PROGRAM MAIN
VAR
	
	hmiAxisSelection: INT := 1; //Not possible to use local hmi variables for array indexes
    afbAxes: ARRAY [1..GVL_APP.nAXIS_NUM] OF FB_Axis;
	
	stAmsNetId	AT %I*	              : AMSNETID;
	nPort	AT %I*                    : WORD;
	nMasterAxisPosition AT %I*        : DINT;
	nMainDriveMarkPosition AT %I*     : DINT;
	nAdditiveTorqueSetpoint    AT %Q* : INT;   // Unit 0.1%  (10=1%)
	dLatchedPosition AT %I*           : DINT;
    fbTemp                            : EL3214_old;
	inputDigSens1 AT %I*              : BOOL;
	inputDigSens2 AT %I*              : BOOL;
	fbModePhase                       : FB_ModePhasing;	 // Phasing Mode
	fbRampVelo                        : FB_RampVelo;
	fbModeVelo                        : FB_ModeVelo;     // Velocity Mode
	fbModePos                         : FB_ModePos;      // Positioning Mode
	fbModeHome                        : FB_ModeHome;     // Homing Mode
	fbIndraDrive                      : fbIndraDrive;    // Control of drive
	
	stCmdEpics                        : ST_CMD_EPICS;    // Control to EPICS 
	stCommands                        : ST_AXIS_COMMAND; // Control to drive
	stStatus                          : ST_AXIS_STATUS;  // Status from drive
	eTargetStateOld                   : TARGET_STATE_MACHINE;
	addStartupTorqueTrigger           : BOOL:=FALSE;
	iTorqueCommandValue  AT %Q*       : INT := 0;
	bApplyTorqueFF                    : BOOL := FALSE;
	nTest: INT;
	
	//hardware
	fbErrorSystem:FB_ErrorSystem;
	fb_s2_EL1809:EL1809;
	fb_s3_EL1809:EL1809;
	fb_s4_EL2819:EL2819;
	fb_s5_EL2819:EL2819;
	fb_s6_EL9505:EL9505;
	fb_s7_EL1252:EL1252;
	fb_s8_EL9410:EL9410;
	fb_s9_EL1252:EL1252;
	fb_s10_EL7201:EL7201;
	fb_s11_EL7201:EL7201;
	fb_s12_EL7201:EL7201;
	fb_s13_EL3214:EL3214;
	fb_s14_EL5021:EL5021;
	fb_s15_EL6695:EL6695;
	fb_s16_EL9410:EL9410;
	fb_s17_EL2032:EL2032;
	fb_s18_EK1110:EK1110;
	fb_s19_IndraDrive:IndraDrive;
	fb_s20_IPOS8020:iPOS8020;
	fb_s21_IPOS8020:iPOS8020;
	fb_s22_IPOS8020:iPOS8020;
	
END_VAR

VAR_INPUT
  stStatEpics                       : ST_STAT_EPICS;   // Status to EPICS
  stHWControlX  : ST_HW_CONTROL_XYZ;
  stHWControlY  : ST_HW_CONTROL_XYZ;
  stHWControlZ  : ST_HW_CONTROL_XYZ;
  stHWControlDev: ST_HW_CONTROL_DEV;
  stHWStatusX   : ST_HW_STATUS_XYZ;
  stHWStatusY   : ST_HW_STATUS_XYZ;
  stHWStatusZ   : ST_HW_STATUS_XYZ;
  stHWStatusDev : ST_HW_STATUS_DEV;
END_VAR

// Check hardware status
ACT_1_Hardware();

// Read Bridge Terminal Inputs
TSCS_Bridge_Inputs();

// Monitor temperature
ACT_2_Temperature();

// Main motor motion
ACT_4_MainDrive();

// Steppers
ACT_5_Steppers();

// Write Bridge Terminal Outputs (incl. test)
TSCS_Bridge_Diagnostic();
TSCS_Bridge_Outputs();

// Error handling
ACT_6_Error();

// Post exe
eTargetStateOld:=stStatEpics.eTargetState;

ACTION ACT_1_Hardware:
// Check state of hardware

// Slave 2 EL1809: General I/O, fuses...
fb_s2_EL1809(ErrorSystem:=fbErrorSystem.pErrorSystem,En:=TRUE,iTerminal_ID:=2);
stHWStatusDev.bEStopOK:=fb_s2_EL1809.bBI_1;                       // s2: ch1: emergency stop ok                 Verify: OK   
stHWStatusDev.bRF02_MainDriveThermalFilterOK:=fb_s2_EL1809.bBI_2; // s2: ch2: rf01 termal braking filter OK..   Verify: Q to Markus: Maybe this should be rd02?
stHWStatusDev.bTA01_TA02_24VSupplyOK:=fb_s2_EL1809.bBI_3;         // s2: ch3: ta01 and ta02 24V power supply OK Verify: OK  
stHWStatusDev.bFC11_Fuse24VOK:=fb_s2_EL1809.bBI_4;                // s2: ch4: fc11 24V fuse OK                   Verify: OK
stHWStatusDev.bFA01_FA02_OvervoltageOK:=fb_s2_EL1809.bBI_5;       // s2: ch5: fa01 and fa02 overvoltage protection OK
stHWStatusDev.bFC01_FuseMainRotationOK:=fb_s2_EL1809.bBI_6;       // s2: ch6: fc01 fuse target wheel motor OK
stHWStatusDev.bFC06_FC07_FuseICSOutletsOK:=fb_s2_EL1809.bBI_7;    // s2: ch7: fc06 and fc07 ICS outlets fuse OK
stHWStatusDev.bFC51_FC52_FC53_FuseUPSOK:=fb_s2_EL1809.bBI_8;      // s2: ch8: fc51, fc52 and fc53 UPS fuses OK (something wrong)

// Slave 3 EL1809: Motion switches (limits)
fb_s3_EL1809(ErrorSystem:=fbErrorSystem.pErrorSystem,En:=TRUE,iTerminal_ID:=3);
main.stHWStatusX.bLimitMax :=fb_s3_EL1809.bBI_1;          // s3: ch1: w02.bg01 stepper x limit max
main.stHWStatusX.bLimitMin :=fb_s3_EL1809.bBI_2;          // s3: ch2: w02.bg02 stepper x limit min
main.stHWStatusX.bLimitMaxMax :=fb_s3_EL1809.bBI_3;       // s3: ch3: w02.bg03 stepper x limit max max
main.stHWStatusX.bLimitMinMin :=fb_s3_EL1809.bBI_4;       // s3: ch4: w02.bg04 stepper x limit min min
main.stHWStatusY.bLimitMax :=fb_s3_EL1809.bBI_5;          // s3: ch5: w02.bg05 stepper y limit max
main.stHWStatusY.bLimitMin :=fb_s3_EL1809.bBI_6;          // s3: ch6: w02.bg06 stepper y limit min
main.stHWStatusY.bLimitMaxMax :=fb_s3_EL1809.bBI_7;       // s3: ch7: w02.bg07 stepper y limit max max
main.stHWStatusY.bLimitMinMin :=fb_s3_EL1809.bBI_8;       // s3: ch8: w02.bg08 stepper y limit min min
main.stHWStatusZ.bLimitMax :=fb_s3_EL1809.bBI_9;          // s3: ch9: w03.bg01 stepper z limit max
main.stHWStatusZ.bLimitMin :=fb_s3_EL1809.bBI_10;         // s3: ch10: w03.bg02 stepper z limit min
main.stHWStatusZ.bLimitMinPark :=fb_s3_EL1809.bBI_11;     // s3: ch11: w03.bg03 stepper z limit min service (lowest switch)
main.stHWStatusZ.bLimitMaxMax :=fb_s3_EL1809.bBI_12;      // s3: ch12: w03.bg04 stepper z limit max max
main.stHWStatusZ.bLimitMinMin :=fb_s3_EL1809.bBI_13;      // s3: ch13: w03.bg05 stepper z limit min min
main.stHWStatusZ.bLimitMinMinPark :=fb_s3_EL1809.bBI_14;  // s3: ch14: w03.bg06 stepper z limit min min service (lowest switch)
main.stHWStatusX.bLimitMinPark:=FALSE;                    // Not used
main.stHWStatusX.bLimitMinMinPark:=FALSE;                 // Not used
main.stHWStatusX.bParkingRangeEnabled:=FALSE;             // Not used;
main.stHWStatusY.bLimitMinPark:=FALSE;                    // Not used
main.stHWStatusY.bLimitMinMinPark:=FALSE;                 // Not used
main.stHWStatusY.bParkingRangeEnabled:=FALSE;             // Not used;

// Slave 4 EL2809: Feed sensors
fb_s4_EL2819(ErrorSystem:=fbErrorSystem.pErrorSystem,En:=TRUE,iTerminal_ID:=4);
stHWControlDev.bRotOmronSensor1Feed:=TRUE;     // s4: ch1: Feed omron sensor 1
stHWControlDev.bRotOmronSensor2Feed:=TRUE;     // s4: ch2: Feed omron sensor 2

// Slave 5 EL2809: Feed switches and brakes
fb_s5_EL2819(ErrorSystem:=fbErrorSystem.pErrorSystem,En:=TRUE,iTerminal_ID:=5);
stHWControlX.bMinMaxFeed:=TRUE;           // s5: ch1: kf05: w02.bg01 w02.bg02 stepper x limit switch max, limit min
//stHWControl.bXBrakeReleaseCmd           // s5: ch2: kf05: w02.ql1: stepper x brake
stHWControlX.bMinMinMaxMaxFeed:=TRUE;     // s5: ch3: kf05: w02.bg03 w02.bg04 stepper x limit switch max max, limit min min
stHWControlY.bMinMaxFeed:=TRUE;           // s5: ch5: kf05: w02.bg05 w02.bg06 stepper y limit switch max, limit min
//stHWControl.bYBrakeReleaseCmd           // s5: ch6: kf05: w02.ql2: stepper y brake
stHWControlY.bMinMinMaxMaxFeed:=TRUE;     // s5: ch7: kf05: w02.bg07 w02.bg08 stepper y limit switch max max, limit min min
stHWControlZ.bMinMaxFeed:=TRUE;           // s5: ch9: kf05: w03.bg01 w03.bg02 w03.bg03  stepper z limit switch max, limit min limit min min (service)
stHWControlZ.bMinMinMaxMaxFeed:=TRUE;     // s5: ch10: kf05: w03.bg04 w03.bg05 w03.bg06  stepper z limit switch max max, limit min min
// Note brakes needs control!!!

// s6: 5V power supply
fb_s6_EL9505(ErrorSystem:=fbErrorSystem.pErrorSystem,En:=TRUE,iTerminal_ID:=6);

// s7: time stamped 5V input from timing system (timing reference pulse 14Hz)
// s7: ch1: kf06. Timing system ref pulse (14Hz). Synch pulse ICS.
fb_s7_EL1252(ErrorSystem:=fbErrorSystem.pErrorSystem,En:=TRUE,iTerminal_ID:=7);

// s8: 24V power supply
fb_s8_EL9410(ErrorSystem:=fbErrorSystem.pErrorSystem,En:=TRUE,iTerminal_ID:=8);

// s9: Omron time stamp 24V
// s9: ch1: w01.bg01 fibre sensor input (home or sector?)
// s9: ch2: w01.bg02 fibre sensor input (home or sector?)
fb_s9_EL1252(ErrorSystem:=fbErrorSystem.pErrorSystem,En:=TRUE,iTerminal_ID:=9);

// s10 ch1: kf09 w02.bg21 Resolver X  
fb_s10_EL7201(ErrorSystem:=fbErrorSystem.pErrorSystem,En:=TRUE,iTerminal_ID:=10);

// s11 ch1: kf10 w02.bg22 Resolver Y
fb_s11_EL7201(ErrorSystem:=fbErrorSystem.pErrorSystem,En:=TRUE,iTerminal_ID:=11);

// s11 ch1: kf11 w03.bg21 Resolver Z
fb_s12_EL7201(ErrorSystem:=fbErrorSystem.pErrorSystem,En:=TRUE,iTerminal_ID:=12);

// s13 EL3214: Temperature inputs X,Y,Z and rotation
fb_s13_EL3214(ErrorSystem:=fbErrorSystem.pErrorSystem,En:=TRUE,iTerminal_ID:=13);
stHWStatusX.fStepperTemp:=INT_TO_LREAL(fb_s13_EL3214.iAI_1)/10; // s13: ch1: kf12 w02.bt01 temperature stepper X PT100
stHWStatusY.fStepperTemp:=INT_TO_LREAL(fb_s13_EL3214.iAI_2)/10; // s13: ch2: kf12 w02.bt02 temperature stepper Y PT100
stHWStatusZ.fStepperTemp:=INT_TO_LREAL(fb_s13_EL3214.iAI_3)/10; // s13: ch3: kf12 w03.bt01 temperature stepper Z PT100
stHWStatusDev.fKF12_RotTemp:=INT_TO_LREAL(fb_s13_EL3214.iAI_4)/10;   // s13: ch4: kf12 Target Main motor Temperature (KTY) (in deg*10)

// s14: Extra encoder (main rotation)
fb_s14_EL5021(ErrorSystem:=fbErrorSystem.pErrorSystem,En:=TRUE,iTerminal_ID:=14);

// s15: Communication to monitoring system
fb_s15_EL6695(ErrorSystem:=fbErrorSystem.pErrorSystem,En:=TRUE,iTerminal_ID:=15);

// s15: 24V power supply
fb_s16_EL9410(ErrorSystem:=fbErrorSystem.pErrorSystem,En:=TRUE,iTerminal_ID:=16);

// s17: MPS com.
fb_s17_EL2032(ErrorSystem:=fbErrorSystem.pErrorSystem,En:=TRUE,iTerminal_ID:=17);

// s1?: Two EL2612 Relay for MPS not in system yet
// s1?: ch1: kf17 Ready for beam
// s1?: ch2: kf17 Beam permit
// s1?: ch3: kf18 Ready for beam
// s1?: ch4: kf18 Beam permit

// s18: extension to drives
fb_s18_EK1110(ErrorSystem:=fbErrorSystem.pErrorSystem,En:=TRUE,iTerminal_ID:=18);

// s19: Main target drive
fb_s19_IndraDrive(ErrorSystem:=fbErrorSystem.pErrorSystem,En:=TRUE,iTerminal_ID:=19);

// s20: Stepper 1
fb_s20_IPOS8020(ErrorSystem:=fbErrorSystem.pErrorSystem,En:=TRUE,iTerminal_ID:=20);

// s21: Stepper 2
fb_s21_IPOS8020(ErrorSystem:=fbErrorSystem.pErrorSystem,En:=TRUE,iTerminal_ID:=21);

// s22: Stepper 3
fb_s22_IPOS8020(ErrorSystem:=fbErrorSystem.pErrorSystem,En:=TRUE,iTerminal_ID:=22);

fbErrorSystem(En:=TRUE);
END_ACTION

ACTION ACT_2_Temperature:
// Function: Monitor tempertures
// Interlock motion on temperatures
// Author: Anders Sandström 2019

stStatEpics.fActTemp:=fb_s13_EL3214.iAI_4/10.0;

// Motor Temperature Monitoring Interlock
IF (stStatEpics.fActTemp >= GVL_Parameters.nMaxMotorTemperature)  OR fbTemp.iAi_Ch1_Stat > 0 THEN
	stCmdEpics.bEnable:= FALSE;
	stCmdEpics.bExecute:= FALSE;
	stStatEpics.nErrorId:=GVL_ErrorCodes.nErrorIndraTempToHigh;
	stStatEpics.sErrorStr:=GVL_ErrorCodes.sErrorIndraTempToHigh;
END_IF
END_ACTION

ACTION ACT_4_MainDrive:

// Enable Axis independent of state (Ensure that drive is ready to enable)
IF stCmdEpics.bEnable THEN
   IF stStatus.bDCBusPresent AND NOT stStatus.bSTOActiveCh1 AND NOT stStatus.bSTOActiveCh2 AND NOT stStatus.bError THEN 
	   stCommands.bEnableAxis :=stCmdEpics.bEnable;
   ELSE
	   stCommands.bEnableAxis := FALSE;
	   stCmdEpics.bExecute := FALSE;
	   stStatEpics.bError:=TRUE;
	   stStatEpics.nErrorId:=GVL_ErrorCodes.nErrorIndraNotReady;
	   stStatEpics.sErrorStr:=GVL_ErrorCodes.sErrorIndraNotReady; 
   END_IF
ELSE
	//Reset enable
    stCommands.bEnableAxis:=stCmdEpics.bEnable;
END_IF

IF stCmdEpics.bExecute THEN
  IF stStatus.bAxisEnabled THEN
    stCommands.bHaltAxis:=stCmdEpics.bExecute;
  ELSE
	stCmdEpics.bExecute:=FALSE;
	stCommands.bHaltAxis:=FALSE;
	stStatEpics.nErrorId:=GVL_ErrorCodes.nErrorNotEnabled;
	stStatEpics.sErrorStr:=GVL_ErrorCodes.sErrorNotEnabled; 
  END_IF
ELSE
  stCommands.bHaltAxis:=stCmdEpics.bExecute;
END_IF

IF NOT stCommands.bEnableAxis THEN
  stCmdEpics.bExecute:=FALSE;
END_IF

stStatEpics.bEnabled:=stStatus.bAxisEnabled;
stCommands.bCmd_ErrorReset:=stCmdEpics.bReset;

stCommands.bCmd_DriveControlledHoming:=FALSE;

// State change
IF stCmdEpics.eTargetStateCmd <> stStatEpics.eTargetState AND NOT stCmdEpics.bexecute AND stStatus.bAxisStandStillStatus THEN
    // Only allow state change if execute is low and at standstill
    stStatEpics.eTargetState:=stCmdEpics.eTargetStateCmd;
END_IF

IF stCmdEpics.fPhaseOffsetMM > GVL_Parameters.fMaxPhaseOffsetMM THEN
	stCmdEpics.fPhaseOffsetMM :=  GVL_Parameters.fMaxPhaseOffsetMM;
END_IF
IF stCmdEpics.fPhaseOffsetMM < GVL_Parameters.fMinPhaseOffsetMM THEN
	stCmdEpics.fPhaseOffsetMM :=  GVL_Parameters.fMinPhaseOffsetMM;
END_IF

stStatEpics.fPhaseOffsetActDeg := stCmdEpics.fPhaseOffsetMM /(GVL_Parameters.fWheelDiameter*pi/360.0);

//nAdditiveTorqueSetpoint:=0;
//IF NOT  stCmdEpics.bExecute THEN
//	addStartupTorqueTrigger:=TRUE;
//END_IF


CASE stStatEpics.eTargetState OF 
	TARGET_STATE_MACHINE.CONSTANT_VELOCITY:
        stCommands.fCommandAcceleration:=GVL_Parameters.fAccDefaultVel;
        stCommands.fCommandDeceleration:=GVL_Parameters.fAccDefaultVel;
		fbModeVelo(
            bExecute:=         stCmdEpics.bExecute,
            bReset:=           stCmdEpics.bReset,
			fVelSet:=          stCmdEpics.fVelSet,
			stStatus:=	       stStatus,	
			stCommands:=       stCommands);
			
			//ramp velocity with selected acceleration
			fbRampVelo(bExecute:=stCmdEpics.bExecute,
              fVelSetIn:=fbModeVelo.fSpeedSetpoint,
              iBlockSampleTimeMicroS:=GVL_Parameters.nTaskSampleTime*1000,
              fVelSetOut:=stCommands.fVelocityCommandValue,
              fVelActIn:=stStatus.fActualVelocity/10);
			  
// add extra torque att startup TEST
		//	IF stStatus.bAxisEnabled AND stCmdEpics.bExecute AND stCmdEpics.fVelSet > 0 THEN
		//		IF stStatus.fActualVelocity/10< stCmdEpics.fVelSet/2 THEN
		//	        nAdditiveTorqueSetpoint:=100;  //Add 10% when under x rpm
		//		ELSIF stStatus.fActualVelocity/10 > stCmdEpics.fVelSet/2 THEN
		//			nAdditiveTorqueSetpoint:=40;
		//		END_IF
		//	END_IF

			
	TARGET_STATE_MACHINE.POSITIONING:
	    stCommands.fCommandAcceleration:=GVL_Parameters.fAccDefaultPos;
        stCommands.fCommandDeceleration:=GVL_Parameters.fAccDefaultPos;

		fbModePos(
            bExecute:=         stCmdEpics.bExecute,
            bReset:=           stCmdEpics.bReset,
			fVelSet:=          stCmdEpics.fVelSet,
			fPosSet:=          stCmdEpics.fPosSet,
			fRefOffset:=       fbModeHome.fActPositionOffset,
			stStatus:=         stStatus,	
			stCommands:=       stCommands);
		
	TARGET_STATE_MACHINE.PHASING:
	    stCommands.fCommandAcceleration:=GVL_Parameters.fAccDefaultVel;
        stCommands.fCommandDeceleration:=GVL_Parameters.fAccDefaultVel;
   		fbModePhase(
			bExecute:=         stCmdEpics.bExecute,
            bReset:=           stCmdEpics.bReset,
			stStatus:=	       stStatus,
			dLatchedPosition:= dLatchedPosition,
			ePhaseType:=       stCmdEpics.ePhaseCntrlAlg,
			ePwmType:=         stCmdEpics.ePhasePwmType,
			stCommands:=       stCommands,
            fPhaseOffsetMM:=   stCmdEpics.fPhaseOffsetMM,
            fRefOffset:=       fbModeHome.fActPositionOffset);
			
			//ramp velocity with selected acceleration (as long as not phasing)
			IF NOT fbModePhase.bPhasing THEN
              fbRampVelo(bExecute:=stCmdEpics.bExecute,
                fVelSetIn:=fbModePhase.fSpeedSetpoint,
                iBlockSampleTimeMicroS:=GVL_Parameters.nTaskSampleTime*1000,
                fVelSetOut:=stCommands.fVelocityCommandValue,
                fVelActIn:=fbModePhase.fLastSectorVelocity);
			ELSE // if phasing then take setpoint direct from fbModePhase
			  stCommands.fVelocityCommandValue:=fbModePhase.fSpeedSetpoint;
            END_IF
						
	TARGET_STATE_MACHINE.HOMING:
        stCommands.fCommandAcceleration:=GVL_Parameters.fAccDefaultVel;
        stCommands.fCommandDeceleration:=GVL_Parameters.fAccDefaultVel;
        fbModeHome( 
            bExecute:=         stCmdEpics.bExecute,
            bReset:=           stCmdEpics.bReset,
			fVelSet:=          GVL_Parameters.fHomeSpeedRpm,
			fPosSet:=          stCmdEpics.fPosSet,
			stStatus:=	       stStatus,	
			stCommands:=       stCommands);
		//stCommands.fFeedrateOverride:=1.0;
		//ramp velocity with selected acceleration
		fbRampVelo(bExecute:=stCmdEpics.bExecute,
              fVelSetIn:=fbModeHome.fSpeedSetpoint,
              iBlockSampleTimeMicroS:=GVL_Parameters.nTaskSampleTime*1000,
              fVelSetOut:=stCommands.fVelocityCommandValue,
              fVelActIn:=stStatus.fActualVelocity/10);
 
	TARGET_STATE_MACHINE.TORQUE:
	    stCommands.fCommandAcceleration:=GVL_Parameters.fAccDefaultVel;
        stCommands.fCommandDeceleration:=GVL_Parameters.fAccDefaultVel;
		stCommands.eOperationMode:=E_OPERATION_MODE_NO.eSecondaryOpMode7;
	    stCommands.eMotionMode :=e_Motion_mode.eJogPositive;
	
	  ELSE  // No valid state
		  
		bApplyTorqueFF:=FALSE;
		stCmdEpics.bExecute:=FALSE;
        stCmdEpics.bEnable:=FALSE;
		stCommands.fVelocityCommandValue:=0;
		stCommands.fCommandVelocity:=0;
		stCommands.fCommandAcceleration:=0;
        stCommands.fCommandDeceleration:=0;
		stStatEpics.nErrorId:=GVL_ErrorCodes.nErrorInvalidState;
	    stStatEpics.sErrorStr:=GVL_ErrorCodes.sErrorInvalidState;
END_CASE

IF bApplyTorqueFF THEN
  // add extra torque att startup TEST
  IF stStatus.bAxisEnabled (*AND stCmdEpics.bExecute*) THEN
	 nAdditiveTorqueSetpoint:=nTest;  //Add 10% when under x rpm
  END_IF
END_IF

IF NOT stCmdEpics.bExecute THEN
	stCommands.fVelocityCommandValue:=0;
END_IF

// TODO: Why I put this here?
//stCommands.eMotionMode:=E_MOTION_MODE.eStop;

// Check maximum velocity
IF stCommands.fCommandVelocity > GVL_Parameters.fMaximumSPeedRpm THEN
  stCommands.fCommandVelocity := GVL_Parameters.fMaximumSPeedRpm;
END_IF
IF stCommands.fVelocityCommandValue > GVL_Parameters.fMaximumSPeedRpm THEN
  stCommands.fVelocityCommandValue := GVL_Parameters.fMaximumSPeedRpm;
END_IF

// Rexroth FB
fbIndraDrive(
	AmsNetId:= stAmsNetId, 
	AdsAddr_Port:= nPort, 
	stAxisCommands:= stCommands, 
	stDriveStatus:= , 
	stAxisStatus=> stStatus, 
	stDriveCommands=> );

// Calculate values for status in EPICS
stStatEpics.fSetVelRaw:= DINT_TO_LREAL(MAIN.fbIndraDrive.stDriveCommands.nS40_VelocityCommandValue)/10000;	
stStatEpics.fActPos:=stStatus.fActualPosition-fbModeHome.fActPositionOffset;
IF stStatEpics.fActPos > 360 THEN
  stStatEpics.fActPos:=stStatEpics.fActPos-360;	
END_IF
IF stStatEpics.fActPos < 0 THEN
  stStatEpics.fActPos:=stStatEpics.fActPos+360;	
END_IF
stStatEpics.fActTorque:=stStatus.fActualTorque;
stStatEpics.fActVel:=stStatus.fActualVelocity/10;
END_ACTION

ACTION ACT_5_Steppers:
// Motion of stepeprs handled in MAIN_NORMAL_MOTION
END_ACTION

ACTION ACT_6_Error:
// Function: Error handling
// Author: Anders Sandström 2019

IF stStatEpics.eTargetState = TARGET_STATE_MACHINE.PHASING THEN
  IF fbModePhase.bError AND NOT stStatEpics.bError THEN
	stStatEpics.bError:=fbModePhase.bError;
	stStatEpics.nErrorId:=fbModePhase.nErrorId;
	stStatEpics.sErrorStr:=fbModePhase.sErrorStr;
  END_IF
  
ELSIF stStatEpics.eTargetState = TARGET_STATE_MACHINE.CONSTANT_VELOCITY THEN
  IF fbModeVelo.bError AND NOT stStatEpics.bError THEN
	stStatEpics.bError:=fbModeVelo.bError;
	stStatEpics.nErrorId:=fbModeVelo.nErrorId;
	stStatEpics.sErrorStr:=fbModeVelo.sErrorStr;
  END_IF
  
ELSIF stStatEpics.eTargetState = TARGET_STATE_MACHINE.POSITIONING THEN
  IF fbModePos.bError AND NOT stStatEpics.bError THEN
	stStatEpics.bError:=fbModePos.bError;
	stStatEpics.nErrorId:=fbModePos.nErrorId;
	stStatEpics.sErrorStr:=fbModePos.sErrorStr;
  END_IF
  
ELSIF stStatEpics.eTargetState = TARGET_STATE_MACHINE.HOMING THEN
  IF fbModeHome.bError AND NOT stStatEpics.bError THEN
    stStatEpics.bError:=fbModeHome.bError;
	stStatEpics.nErrorId:=fbModeHome.nErrorId;
	stStatEpics.sErrorStr:=fbModeHome.sErrorStr;
  END_IF
END_IF

// To high velocity detected. Shutdown..
IF ABS(stStatus.fActualVelocity)/10 > GVL_Parameters.fMaximumSPeedRpm THEN 
  stCommands.bEnableAxis:= FALSE;
  stCmdEpics.bEnable:=FALSE;
  stCmdEpics.bExecute:=FALSE;
  stStatEpics.bError:=TRUE;
  stStatEpics.nErrorId:=GVL_ErrorCodes.nErrorVelToHigh;
  stStatEpics.sErrorStr:=GVL_ErrorCodes.sErrorVelToHigh;
END_IF

IF stcmdEpics.bReset THEN
  stStatEpics.bError:=FALSE;
  stStatEpics.nErrorId:=GVL_ErrorCodes.nErrorCodeOKId;
  stStatEpics.sErrorStr:=GVL_ErrorCodes.nErrorCodeOKStr;
  stStatEpics.bBrake1TempAlarm:=FALSE;
  stStatEpics.bBrake2TempAlarm:=FALSE;
END_IF
stcmdEpics.bReset:=FALSE;
END_ACTION

ACTION ACT_X_Diag:
// Function: Some parameters just for debugging
// Note: Do not need to be executed, can be watched online anyway..
// Author: Anders Sandström 2019

	stCommands.bCmd_ActivateParameterMode;//True puts the drive in parameter mode
	stCommands.bCmd_DisableLimits;// True disables monitoring of errors
	stCommands.bCmd_DriveControlledHoming;// True starts homing procedure defined in the drive
	stCommands.bCmd_ErrorReset;
	stCommands.bCmd_ExitParameterMode;
	stCommands.bCmd_RunVirtualMater;// Jog command to the virtual master
	stCommands.bCmd_SetAbsolutePosition;
	stCommands.bCommandPositionChange;// Drive moves to the current target position, when bCommandVAlueAccept toggled, drive moves to the new target position
	stCommands.bCommandValueAccept;// Used in "Drive positioning Mode" to update the target position when toggled
	stCommands.bEnableAxis;
	stCommands.bHaltAxis;// Performs halt on the drive, bEnableaxis has to be TRUE
	stCommands.bPositionCommandValue;//0=Absolute;1=Relative
	stCommands.eMotionMode;
	stCommands.eOperationMode;
	stCommands.fCommandAcceleration;// Acceleration used for positioning and jogging
	stCommands.fCommandDeceleration;// Deceleration used for positioning and jogging
	stCommands.fCommandPosition;
	stCommands.fCommandVelocity;// Velocity used for positioning and jogging
	stCommands.fFeedrateOverride;// Parameter used for adjustment of the velocity (0,100)%
	stCommands.fTorqueLimit;
	stCommands.fVelocityCommandValue;// S40, velocity used for positining and jogging (in velocity mode)
	stStatus.bAxisEnabled;
END_ACTION

END_PROGRAM

(* stored: Version 1.1.0.1, ProductVersion 3.1.4024.6
   POU MAIN: Id {40828a63-f1c1-40a3-a7c5-8a47be350a36}, SpecialFunc None
   Action ACT_1_Hardware: Id {713eae55-748e-42a3-b2f0-81f54e66f4bd}
   Action ACT_2_Temperature: Id {ec2bd795-c2d7-49be-acd7-2671eaea481b}
   Action ACT_4_MainDrive: Id {0608089f-ed53-4fbf-a585-99ff0324bc84}
   Action ACT_5_Steppers: Id {3a068380-4e98-46e5-9ef4-f9271d802bcf}
   Action ACT_6_Error: Id {6316e704-a716-4c28-824a-a22fe5448145}
   Action ACT_X_Diag: Id {2a0ea7d8-8ff8-4796-ae8a-6c3ebb6f7955} *)
